(* CODESYS project Assigment1.export

Project tree, tasks and I/O mapping:
  control/
    function block CylinderFB [LD]
    program cylinder_ctrl [LD]
    program cylinder_ctrl_SFC [LD]
    program fbd_ctrl [FBD]
    function block LampCTRL [SFC]
    function block Sequence [SFC]
*)

// control/CylinderFB
FUNCTION_BLOCK CylinderFB
VAR_INPUT
	extend: BOOL;
	retract: BOOL;
	cyl_in: BOOL;
	cyl_out: BOOL;
	delay: TIME;
END_VAR
VAR_OUTPUT
	ctrl: BOOL;
	count: INT:=0;
END_VAR
VAR
	TOF_0: TOF;
	TOF_1: TOF;
	delay_close: TON;
END_VAR
VAR // added by the converter: edge detectors and wires of the graphical bodies
    _rt1, _rt2 : R_TRIG;
END_VAR

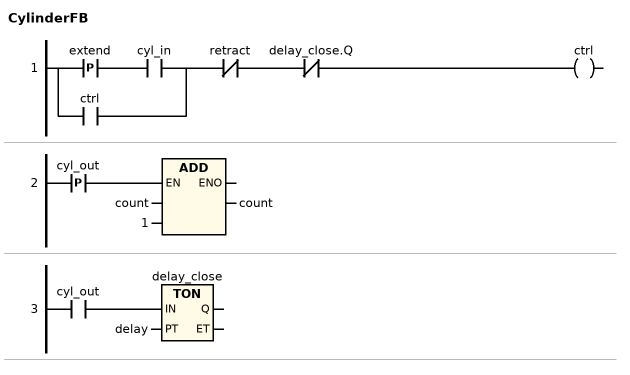
// NETWORK 1
_rt1(CLK := extend);
ctrl := (_rt1.Q AND cyl_in OR ctrl) AND NOT retract AND NOT delay_close.Q;

// NETWORK 2
_rt2(CLK := cyl_out);
IF _rt2.Q THEN count := count + 1; END_IF

// NETWORK 3
delay_close(IN := cyl_out, PT := delay); // TON

END_FUNCTION_BLOCK

// control/cylinder_ctrl
PROGRAM cylinder_ctrl
VAR
    Cylinder1: CylinderFB;
    Cylinder2: CylinderFB;
    Cylinder3: CylinderFB;
    starting: BOOL :=FALSE;
    init: BOOL :=TRUE;
	init_23: BOOL :=FALSE;
    cyl_1_out: BOOL :=FALSE;
    cyl_1_done: BOOL :=FALSE;
	cyl_23_out: BOOL:=FALSE;
	cyl_23_done: BOOL:=FALSE;
	LampCTRL: LampCTRL;
END_VAR
VAR // added by the converter: edge detectors and wires of the graphical bodies
    _rt1 : R_TRIG;
    _w1, _w2, _w3, _w4, _w5 : BOOL;
    _ft1 : F_TRIG;
END_VAR

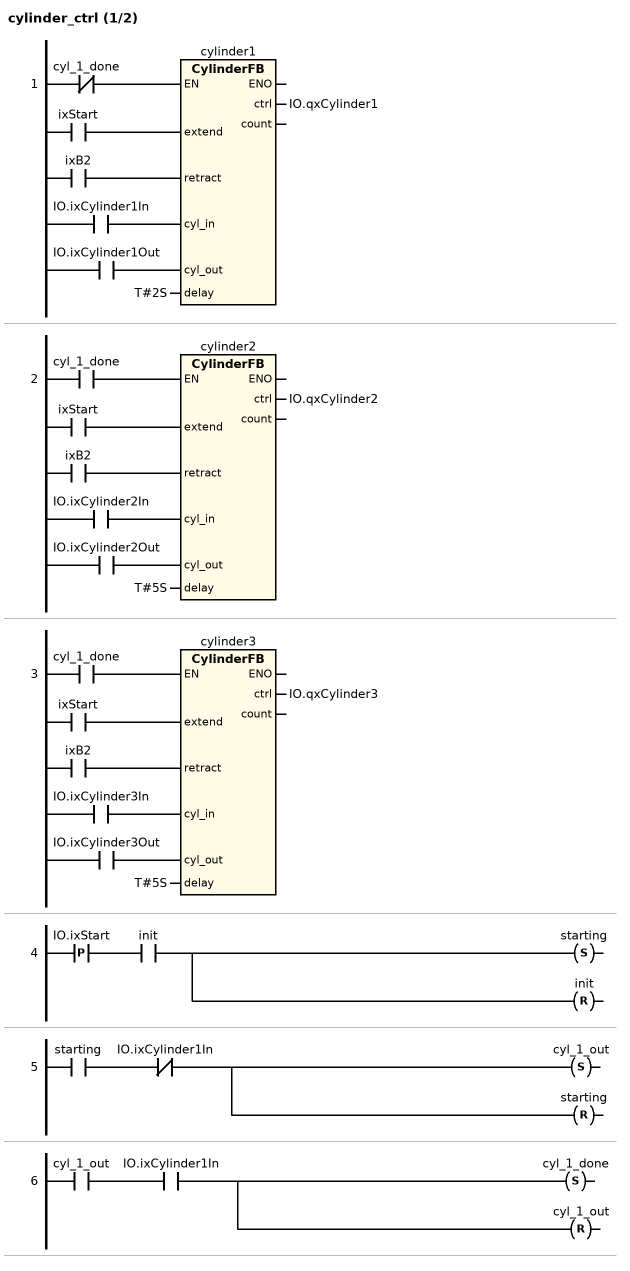
// NETWORK 1
IF NOT cyl_1_done THEN
    cylinder1(
        extend := ixStart,
        retract := ixB2,
        cyl_in := IO.ixCylinder1In,
        cyl_out := IO.ixCylinder1Out,
        delay := T#2S,
        ctrl => IO.qxCylinder1); // CylinderFB
END_IF

// NETWORK 2
IF cyl_1_done THEN
    cylinder2(
        extend := ixStart,
        retract := ixB2,
        cyl_in := IO.ixCylinder2In,
        cyl_out := IO.ixCylinder2Out,
        delay := T#5S,
        ctrl => IO.qxCylinder2); // CylinderFB
END_IF

// NETWORK 3
IF cyl_1_done THEN
    cylinder3(
        extend := ixStart,
        retract := ixB2,
        cyl_in := IO.ixCylinder3In,
        cyl_out := IO.ixCylinder3Out,
        delay := T#5S,
        ctrl => IO.qxCylinder3); // CylinderFB
END_IF

// NETWORK 4
_rt1(CLK := IO.ixStart);
_w1 := _rt1.Q AND init;
starting S= _w1;
init R= _w1;

// NETWORK 5
_w2 := starting AND NOT IO.ixCylinder1In;
cyl_1_out S= _w2;
starting R= _w2;

// NETWORK 6
_w3 := cyl_1_out AND IO.ixCylinder1In;
cyl_1_done S= _w3;
cyl_1_out R= _w3;

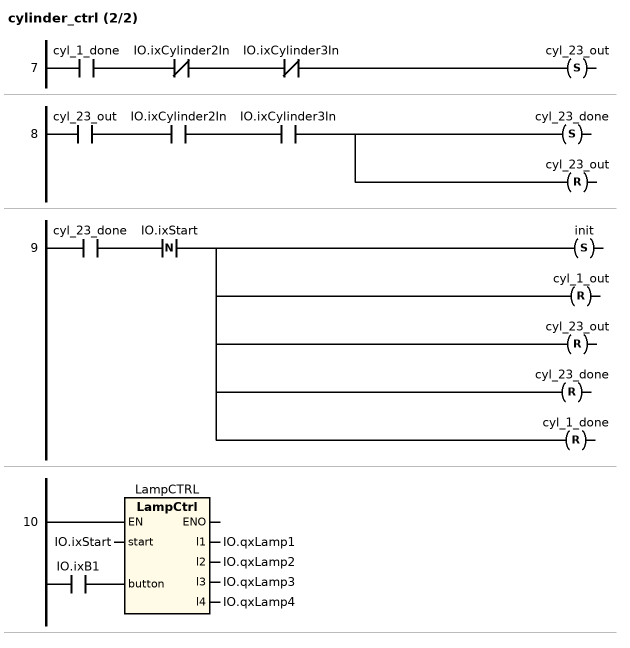
// NETWORK 7
cyl_23_out S= cyl_1_done AND NOT IO.ixCylinder2In AND NOT IO.ixCylinder3In;

// NETWORK 8
_w4 := cyl_23_out AND IO.ixCylinder2In AND IO.ixCylinder3In;
cyl_23_done S= _w4;
cyl_23_out R= _w4;

// NETWORK 9
_ft1(CLK := IO.ixStart);
_w5 := cyl_23_done AND _ft1.Q;
init S= _w5;
cyl_1_out R= _w5;
cyl_23_out R= _w5;
cyl_23_done R= _w5;
cyl_1_done R= _w5;

// NETWORK 10
LampCTRL(
    start := IO.ixStart,
    button := IO.ixB1,
    l1 => IO.qxLamp1,
    l2 => IO.qxLamp2,
    l3 => IO.qxLamp3,
    l4 => IO.qxLamp4);

END_PROGRAM

// control/LampCTRL
FUNCTION_BLOCK LampCTRL
VAR_INPUT
	start: BOOL;
	button: BOOL;
END_VAR
VAR_OUTPUT
	l1: BOOL;
	l2: BOOL;
	l3: BOOL;
	l4: BOOL;
END_VAR
VAR
END_VAR

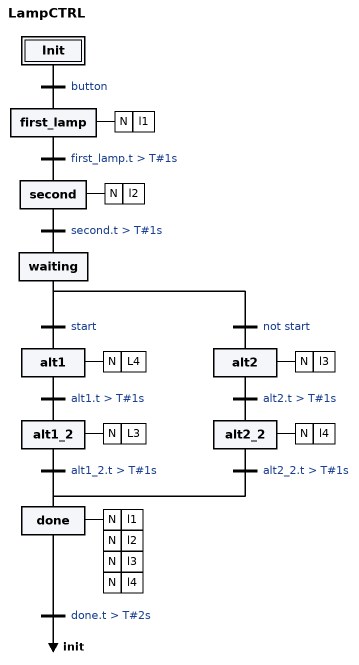
INITIAL_STEP Init:
END_STEP
TRANSITION FROM Init TO first_lamp
    := button;
END_TRANSITION
STEP first_lamp:
    l1(N);
END_STEP
TRANSITION FROM first_lamp TO second
    := first_lamp.t > T#1s;
END_TRANSITION
STEP second:
    l2(N);
END_STEP
TRANSITION FROM second TO waiting
    := second.t > T#1s;
END_TRANSITION
STEP waiting:
END_STEP
TRANSITION FROM waiting TO alt1
    := start;
END_TRANSITION
STEP alt1:
    L4(N);
END_STEP
TRANSITION FROM alt1 TO alt1_2
    := alt1.t > T#1s;
END_TRANSITION
STEP alt1_2:
    L3(N);
END_STEP
TRANSITION FROM alt1_2 TO done
    := alt1_2.t > T#1s;
END_TRANSITION
TRANSITION FROM waiting TO alt2
    := not start;
END_TRANSITION
STEP alt2:
    l3(N);
END_STEP
TRANSITION FROM alt2 TO alt2_2
    := alt2.t > T#1s;
END_TRANSITION
STEP alt2_2:
    l4(N);
END_STEP
TRANSITION FROM alt2_2 TO done
    := alt2_2.t > T#1s;
END_TRANSITION
STEP done:
    l1(N);
    l2(N);
    l3(N);
    l4(N);
END_STEP
TRANSITION FROM done TO init
    := done.t > T#2s;
END_TRANSITION

END_FUNCTION_BLOCK

// control/cylinder_ctrl_SFC
PROGRAM cylinder_ctrl_SFC
VAR
    Cylinder1: CylinderFB;
    Cylinder2: CylinderFB;
    Cylinder3: CylinderFB;
    starting: BOOL :=FALSE;
    init: BOOL :=TRUE;
	init_23: BOOL :=FALSE;
    cyl_1_out: BOOL :=FALSE;
    cyl_1_done: BOOL :=FALSE;
	cyl_23_out: BOOL:=FALSE;
	cyl_23_done: BOOL:=FALSE;
	LampCTRL: LampCTRL;
	sequence_ctrl: Sequence;
	r_trig:R_TRIG;
	count: INT;
END_VAR

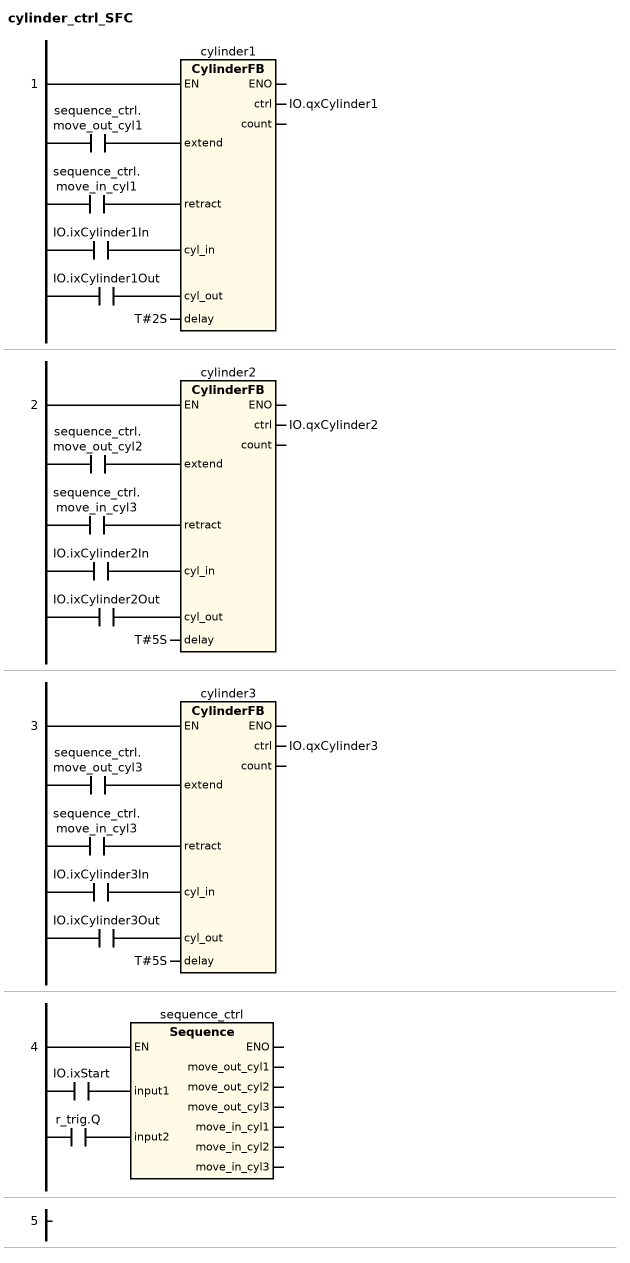
// NETWORK 1
cylinder1(
    extend := sequence_ctrl.move_out_cyl1,
    retract := sequence_ctrl.move_in_cyl1,
    cyl_in := IO.ixCylinder1In,
    cyl_out := IO.ixCylinder1Out,
    delay := T#2S,
    ctrl => IO.qxCylinder1); // CylinderFB

// NETWORK 2
cylinder2(
    extend := sequence_ctrl.move_out_cyl2,
    retract := sequence_ctrl.move_in_cyl3,
    cyl_in := IO.ixCylinder2In,
    cyl_out := IO.ixCylinder2Out,
    delay := T#5S,
    ctrl => IO.qxCylinder2); // CylinderFB

// NETWORK 3
cylinder3(
    extend := sequence_ctrl.move_out_cyl3,
    retract := sequence_ctrl.move_in_cyl3,
    cyl_in := IO.ixCylinder3In,
    cyl_out := IO.ixCylinder3Out,
    delay := T#5S,
    ctrl => IO.qxCylinder3); // CylinderFB

// NETWORK 4
sequence_ctrl(input1 := IO.ixStart, input2 := r_trig.Q); // Sequence

// NETWORK 5

END_PROGRAM

// control/Sequence
FUNCTION_BLOCK Sequence
VAR_INPUT
	input1: BOOL;
	input2: BOOL;
END_VAR
VAR_OUTPUT
	move_out_cyl1: BOOL;
	move_out_cyl2: BOOL;
	move_out_cyl3: BOOL;
	move_in_cyl1: BOOL;
	move_in_cyl2: BOOL;
	move_in_cyl3: BOOL;
END_VAR
VAR
END_VAR

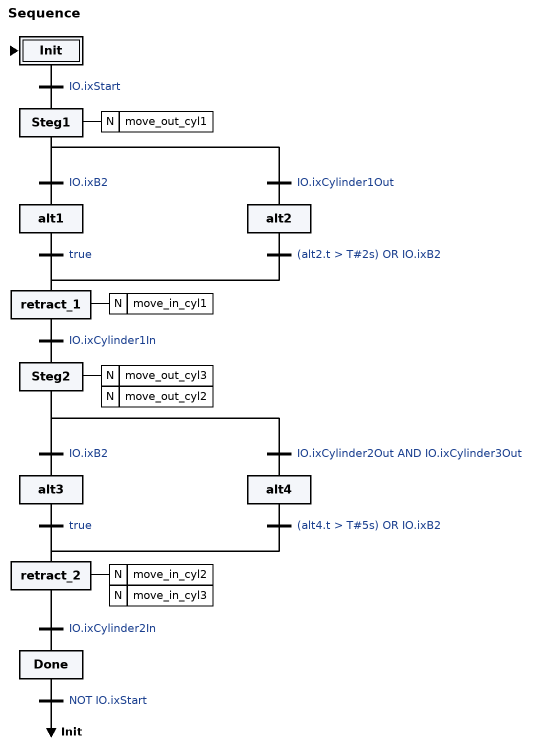
INITIAL_STEP Init:
END_STEP
TRANSITION FROM Init TO Steg1
    := IO.ixStart;
END_TRANSITION
STEP Steg1:
    move_out_cyl1(N);
END_STEP
TRANSITION FROM Steg1 TO alt1
    := IO.ixB2;
END_TRANSITION
STEP alt1:
END_STEP
TRANSITION FROM alt1 TO retract_1
    := true;
END_TRANSITION
TRANSITION FROM Steg1 TO alt2
    := IO.ixCylinder1Out;
END_TRANSITION
STEP alt2:
END_STEP
TRANSITION FROM alt2 TO retract_1
    := (alt2.t > T#2s) OR IO.ixB2;
END_TRANSITION
STEP retract_1:
    move_in_cyl1(N);
END_STEP
TRANSITION FROM retract_1 TO Steg2
    := IO.ixCylinder1In;
END_TRANSITION
STEP Steg2:
    move_out_cyl3(N);
    move_out_cyl2(N);
END_STEP
TRANSITION FROM Steg2 TO alt3
    := IO.ixB2;
END_TRANSITION
STEP alt3:
END_STEP
TRANSITION FROM alt3 TO retract_2
    := true;
END_TRANSITION
TRANSITION FROM Steg2 TO alt4
    := IO.ixCylinder2Out AND IO.ixCylinder3Out;
END_TRANSITION
STEP alt4:
END_STEP
TRANSITION FROM alt4 TO retract_2
    := (alt4.t > T#5s) OR IO.ixB2;
END_TRANSITION
STEP retract_2:
    move_in_cyl2(N);
    move_in_cyl3(N);
END_STEP
TRANSITION FROM retract_2 TO Done
    := IO.ixCylinder2In;
END_TRANSITION
STEP Done:
END_STEP
TRANSITION FROM Done TO Init
    := NOT IO.ixStart;
END_TRANSITION

END_FUNCTION_BLOCK

// control/fbd_ctrl
PROGRAM fbd_ctrl
VAR
END_VAR

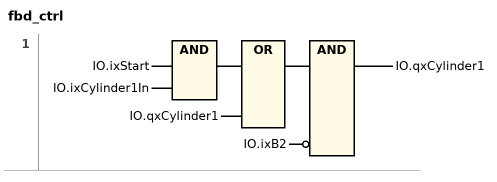
// NETWORK 1
IO.qxCylinder1 := (IO.ixStart AND IO.ixCylinder1In OR IO.qxCylinder1) AND NOT IO.ixB2;

END_PROGRAM
